// TIA Portal V20 export
// export: Created 2025-12-01T14:56:19.2090589Z, ExportSetting None, DisplayName Totally Integrated Automation Portal, DisplayVersion V20 Update 3, DisplayName TIA Portal Openness, DisplayVersion V20 Update 3, DisplayName TIA Portal Version Control Interface, DisplayVersion V20 Update 3, DisplayName STEP 7 Professional, DisplayVersion V20 Update 3, DisplayName STEP 7 Safety, DisplayVersion V20 Update 2, DisplayName WinCC Basic/Comfort/Advanced, DisplayVersion V20 Update 3, DisplayName WinCC Professional, DisplayVersion V20 Update 3, DisplayName WinCC Unified, DisplayVersion V20 Update 3
TYPE "i950 Estatus variador"
   STRUCT
      "Ready For Operation" : Bool;
      "Homing Busy" : Bool;
      "Operation Enabled" : Bool;
      "Drive Fault" : Bool;
      "Drive Homed" : Bool;
      "Quickstop Active" : Bool;
      "Jogging Busy" : Bool;
      "Drive Warning" : Bool;
      "Halt Busy" : Bool;
      "Motorcontrol limited" : Bool;
      "Target Reached" : Bool;
      "Abort Busy" : Bool;
      Standstill : Bool;
      "Direction Negative" : Bool;
      "Brake Released" : Bool;
      "STO Active" : Bool;
      "Profile No 01 Active" : Bool;
      "Profile No 02 Active" : Bool;
      "Profile No 04 Active" : Bool;
      "Profile No 08 Active" : Bool;
      "Positioning Profile Done" : Bool;
      "Limit Switch Negative" : Bool;
      "Limit Switch Positive" : Bool;
      "Touch Probe Home Switch" : Bool;
      "Status Signal Bit 25" : Bool;
      "Status Signal Bit 26" : Bool;
      "Torque setpoint limited" : Bool;
      "External Position Active" : Bool;
      "External Velocity Active" : Bool;
      "External Acc Dec Jerk Active" : Bool;
      "External ToqueLimit Active" : Bool;
   END_STRUCT;
END_TYPE
